{attribute addProperty BoxType "EP4374-0002-0016"}
{attribute addProperty Id "AI_TxPDO_Map_Standard_ChannelAT %I*ARRAY[0..1] OF AI_TxPDO_Map_Standard_Channel_087F71C76480AO_RxPDO_Map_ChannelAT %Q*ARRAY[0..1] OF AO_RxPDO_Map_Channel_F57FA4F93240WcStateAT %I*WcState_F855686C1620InfoDataAT %I*InfoData_BC63D37F80100"}
{attribute addProperty CRC "84439475"}
{attribute addProperty SizeInBites "192"}
{attribute addProperty SizeInBytes "24"}
TYPE EP4374_55F35795 :
STRUCT
	{attribute addProperty Name "AI_TxPDO_Map_Standard_Channel"}
	AI_TxPDO_Map_Standard_Channel : ARRAY[0..1] OF AI_TxPDO_Map_Standard_Channel_087F71C7;
	{attribute addProperty Name "AO_RxPDO_Map_Channel"}
	AO_RxPDO_Map_Channel : ARRAY[0..1] OF AO_RxPDO_Map_Channel_F57FA4F9;
	{attribute addProperty Name "WcState"}
	WcState : WcState_F855686C;
	{attribute addProperty Name "InfoData"}
	InfoData : InfoData_BC63D37F;
END_STRUCT
END_TYPE

(* stored: Version 1.2.0.0, ProductVersion 3.1.4024.9
   DUT EP4374_55F35795: Id {8538ea4c-f85f-460f-bff5-0584d1981f9c} *)
